(* Logix 5000 project; controller Commerford_topping_5477_V3 vendor 1 type 14 code 222 rev 33.11; software revision 33.02; part 2 of 6 *)
(* tags used below, declared in another part *)
   PackTags : PACKMLv30;
   Sts_Clearing : BOOL;   // Clearing
   Sts_Starting : BOOL;   // Starting
   Sts_Execute : BOOL;   // Execute
   Sts_Stopping : BOOL;   // Stopping
   Sts_Aborting : BOOL;   // Aborting
   Sts_Holding : BOOL;   // Holding
   Sts_Unholding : BOOL;   // Unholding
   Sts_Suspending : BOOL;   // Suspending
   Sts_Unsuspending : BOOL;   // Unsuspending
   Sts_Resetting : BOOL;   // Resetting
   Sts_Completing : BOOL;   // Completing
   Process_Selected : SINT;   // Recipe number selects which PackTag.command.product[#] will be used.
   Sts_MachineFaulted : BOOL;   // Machine recieved an fault trigger
   Sts_ProcessActive : BOOL;   // Machine is running a process.
   Reset_Signal : BOOL;   // Reset signal to EMs
   MachineState : USINT;   // Technical Report Equipment States: 1 Clearing 2 Stopped 3 Starting 4 Idle 5 Suspended 6 Execute 7 Stopping 8 Aborting 9
   wrk_compare_UDINT : UDINT;
   i : DINT;   // index num, only for local use. used for forloops
   wrk_prev_state : DINT;   // local mem
   wrk_SwitchLayer_To_Maintenance : DINT;
   wrk_SwitchLayer_To_Manual : DINT;
   wrk_SwitchLayer_To_Automatic : DINT;
(* ISA_TR_88_00_02, continued *)

ROUTINE Prescan   (* structured text *)
// Clear old mem
   ////////////////////////////////////////////////////////////
   //   Copyright (c)
   //------------------------------------------------------------
   //   Routine: Prescan
   //   Author: WPI\tom.reit
   //   Created: 2-11-2022
   //------------------------------------------------------------
   //   Description:
   //           Clear old mem
   //
   //
   //   History:
   //
   ////////////////////////////////////////////////////////////
   
   wrk_compare_UDINT:=0;
   for i := 0 to 31 do
   	wrk_compare_UDINT:=(1*2**i)+wrk_compare_UDINT;	// set compare value, cant move 64bits so have to do some clever bit manipulation.
   end_for;
   
   
   wrk_prev_state						:=	-1;					// set mem state to something that machineState can never be. therfor the whileloop will always execute
   MachineState						:=	9;					// always start safe, in aborted.
   Sts_MachineFaulted					:=	1;					// Machine is always faulted on startup from cold start.
   PackTags.Status.StateRequested		:=	MachineState;		// Set requested state same as actual state.
   
   wrk_SwitchLayer_To_Maintenance		:=0;		// Set layer switching to begin step.
   wrk_SwitchLayer_To_Manual			:=0;		// Set layer switching to begin step.
   wrk_SwitchLayer_To_Automatic		:=0;		// Set layer switching to begin step.
   
   Process_Selected					:=1;		// always run with first recipe on start.
   
   /* Reset ModeCumulativeTime for admin tags */
   for i := 0 to 6 do
   	PackTags.Admin.ModeCumulativeTime[i]:=0;
   end_for;
   
   Sts_ProcessActive:=0;
   
END_ROUTINE
END_ADD_ON_INSTRUCTION

ADD_ON_INSTRUCTION ISA_TR_88_00_02_StateChangeRequest   (* revision 1.0, ExecutePrescan, ExecuteEnableInFalse *)
VAR_IN_OUT
   Packml : PACKMLv30; {required}
END_VAR
VAR_INPUT
   RequestCmd : USINT; {required}   // 0 Undefined 1 Reset 2 Start 3 Stop 4 Hold 5 Unhold 6 Suspend 7 Unsuspend 8 Abort 9 Clear
END_VAR
VAR_OUTPUT
   Sts_StateTransition_Succesfull : BOOL; {access Read Only, visible}
   Sts_StateTransition_Failed : BOOL; {access Read Only, visible}
END_VAR
VAR
   dstepnum : DINT; {access None}
   Wrk_requestedState : DINT; {access None}
   ValidRequest : BOOL; {access None}   // check if request is valid
END_VAR

ROUTINE EnableInFalse   (* structured text *)
   ////////////////////////////////////////////////////////////
   //   Copyright (c)
   //------------------------------------------------------------
   //   Routine: EnableInFalse
   //   Author: WPI\tom.reit
   //   Created: 25-5-2023
   //------------------------------------------------------------
   //   Description:
   //
   //
   //   History:
   //
   ////////////////////////////////////////////////////////////
   dstepnum							:=0;
   Sts_StateTransition_Succesfull		:=0;
   Sts_StateTransition_Failed			:=0;
END_ROUTINE

ROUTINE Logic   (* structured text *)
   ////////////////////////////////////////////////////////////
   //   Copyright (c)
   //------------------------------------------------------------
   //   Routine: ISA_TR_88_00_02_StateChangeRequest - Logic
   //   Author: WPI\tom.reit
   //   Created: 24-5-2023
   //------------------------------------------------------------
   //   Description:
   //
   //
   //   History:
   //
   ////////////////////////////////////////////////////////////
   if dstepnum=0 AND EnableIn then
   	Sts_StateTransition_Succesfull		:=0;
   	Sts_StateTransition_Failed			:=0;
   	dstepnum:=1;
   end_if;
   case dstepnum of
   	1: /* send Unit command */
   		ValidRequest					:=0;
   		Packml.Command.CntrlCmd			:=RequestCmd;
   		Packml.Command.CmdChangeRequest	:=1;
   		case RequestCmd of
   			0:/* Undefined */
   			1:/* Reset */
   				if Packml.Status.StateCurrent = 2 then ValidRequest:=1; end_if;
   			2:/* Start */
   				if Packml.Status.StateCurrent = 4 then ValidRequest:=1; end_if;
   			3:/* Stop */
   				if Packml.Status.StateCurrent <> 8 then ValidRequest:=1; end_if;
   				if Packml.Status.StateCurrent <> 9 then ValidRequest:=1; end_if;
   				if Packml.Status.StateCurrent <> 1 then ValidRequest:=1; end_if;
   			4:/* Hold */
   				if Packml.Status.StateCurrent = 6 then ValidRequest:=1; end_if;
   			5:/* Unhold */
   				if Packml.Status.StateCurrent = 11 then ValidRequest:=1; end_if;
   			6:/* Suspend */
   				if Packml.Status.StateCurrent = 6 then ValidRequest:=1; end_if;
   			7:/* Unsuspend */
   				if Packml.Status.StateCurrent = 5 then ValidRequest:=1; end_if;
   			8:/* Abort */
   				ValidRequest:=1;
   			9:/* Clear */
   				if Packml.Status.StateCurrent = 9 then ValidRequest:=1; end_if;
   			10:/* Complete */
   				if Packml.Status.StateCurrent = 6 then ValidRequest:=1; end_if;
   			else
   		end_case;
   		dstepnum						:=2;
   	2: /* Acknowledge Unit Status, machine recieved command. */
   		if ValidRequest then
   			dstepnum						:=3;
   		else
   			dstepnum						:=999;
   		end_if;
   	3: /* Acknowledge Unit Status, machine recieved command. */
   		if NOT Packml.Command.CmdChangeRequest then
   			dstepnum						:=1000;
   		end_if;
   	999:/* Failed */
   		Sts_StateTransition_Succesfull		:=0;
   		Sts_StateTransition_Failed			:=1;
   	1000:/* Succesfull */
   		Sts_StateTransition_Succesfull		:=1;
   		Sts_StateTransition_Failed			:=0;
   	else
   		dstepnum:=0;
   end_case;
   
END_ROUTINE

ROUTINE Prescan   (* structured text *)
   ////////////////////////////////////////////////////////////
   //   Copyright (c)
   //------------------------------------------------------------
   //   Routine: Prescan
   //   Author: WPI\tom.reit
   //   Created: 25-5-2023
   //------------------------------------------------------------
   //   Description:
   //
   //
   //   History:
   //
   ////////////////////////////////////////////////////////////
   dstepnum							:=0;
   Sts_StateTransition_Succesfull		:=0;
   Sts_StateTransition_Failed			:=0;
END_ROUTINE
END_ADD_ON_INSTRUCTION

ADD_ON_INSTRUCTION ProcessHandler   (* revision 1.0, vendor WPI *)
VAR_IN_OUT
   PackML : ISA_TR_88_00_02; {required}
   bStateTransitions : DINT[32]; {required}
END_VAR
VAR_OUTPUT
   Sts_Unsuspending_PC : BOOL; {access Read Only}
   Sts_Unholding_PC : BOOL; {access Read Only}
   Sts_SuspendTrigger : BOOL; {access Read Only}
   Sts_Suspending_PC : BOOL; {access Read Only}
   Sts_Stopping_PC : BOOL; {access Read Only}
   Sts_Starting_PC : BOOL; {access Read Only}
   Sts_Resetting_PC : BOOL; {access Read Only}
   Sts_Holding_PC : BOOL; {access Read Only}
   Sts_Force_Stop : BOOL; {access Read Only}
   Sts_Force_Abort : BOOL; {access Read Only}
   Sts_Faulted : BOOL; {access Read Only}
   Sts_Executing : BOOL; {access Read Only}
   Sts_Process_Selected : BOOL; {access Read Only, visible}
   Sts_Completing_PC : BOOL; {access Read Only}
   Sts_Clearing_PC : BOOL; {access Read Only}
   Sts_Aborting_PC : BOOL; {access Read Only}
   OwnershipFault : BOOL; {access Read Only, visible}
END_VAR
VAR_INPUT
   Select : BOOL; {visible}   // Selecting Process will incuding in Unit state transitions
END_VAR
VAR_IN_OUT
   ProcessModule : ProcessModule; {required}
END_VAR
VAR_INPUT
   Process_ID : USINT; {required}
END_VAR
VAR
   UnasignOwnership : BOOL; {access None}
   AsignOwnership : BOOL; {access None}
END_VAR

ROUTINE Logic   (* ladder *)
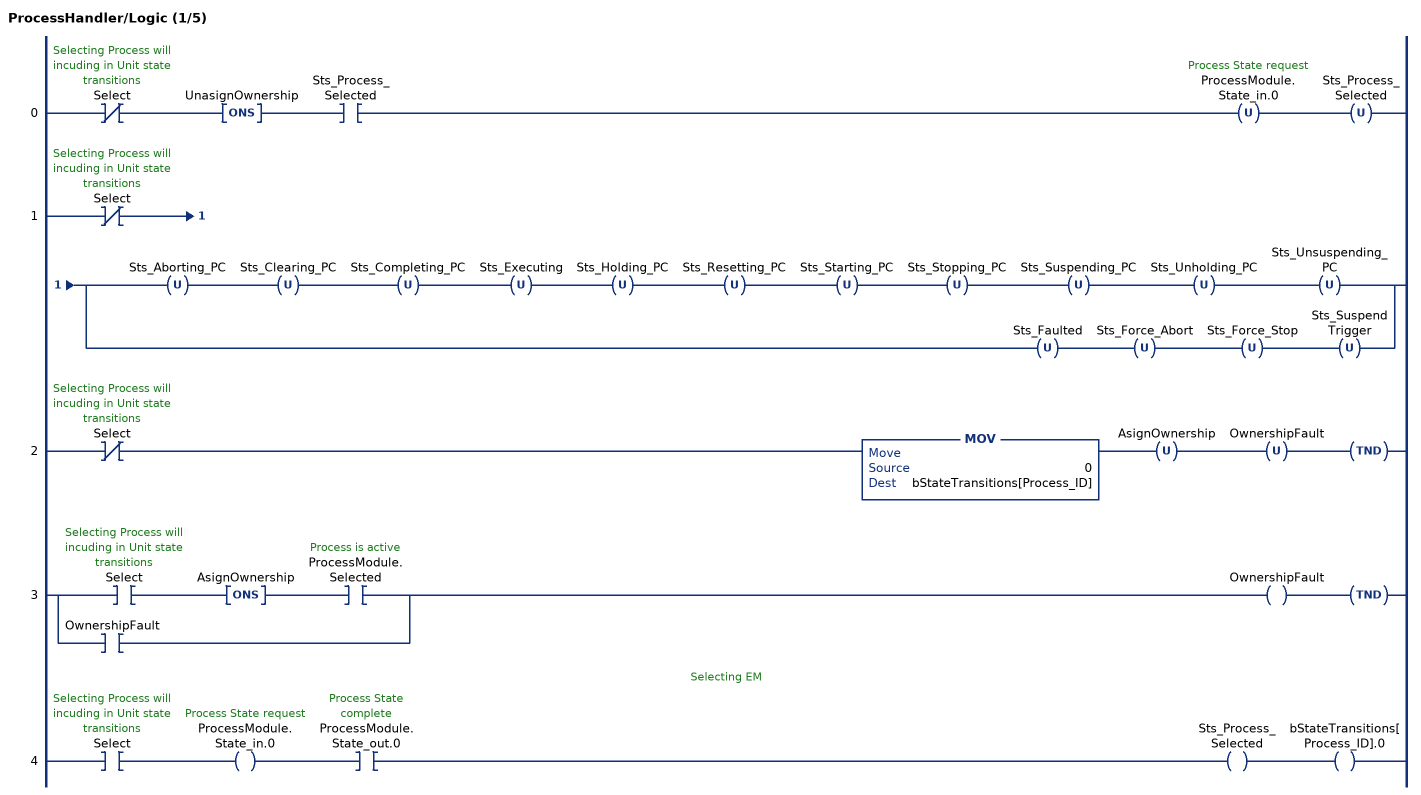
   0: XIO(Select)ONS(UnasignOwnership)XIC(Sts_Process_Selected)OTU(ProcessModule.State_in.0)OTU(Sts_Process_Selected);
   1: XIO(Select)[OTU(Sts_Aborting_PC) OTU(Sts_Clearing_PC) OTU(Sts_Completing_PC) OTU(Sts_Executing) OTU(Sts_Holding_PC) OTU(Sts_Resetting_PC) OTU(Sts_Starting_PC) OTU(Sts_Stopping_PC) OTU(Sts_Suspending_PC) OTU(Sts_Unholding_PC) OTU(Sts_Unsuspending_PC) ,OTU(Sts_Faulted) OTU(Sts_Force_Abort) OTU(Sts_Force_Stop) OTU(Sts_SuspendTrigger) ];
   2: XIO(Select)MOV(0,bStateTransitions[Process_ID])OTU(AsignOwnership)OTU(OwnershipFault)TND();
   3: [XIC(Select) ONS(AsignOwnership) XIC(ProcessModule.Selected) ,XIC(OwnershipFault) ]OTE(OwnershipFault)TND();
   // Selecting EM
   4: XIC(Select)OTE(ProcessModule.State_in.0)XIC(ProcessModule.State_out.0)OTE(Sts_Process_Selected)OTE(bStateTransitions[Process_ID].0);
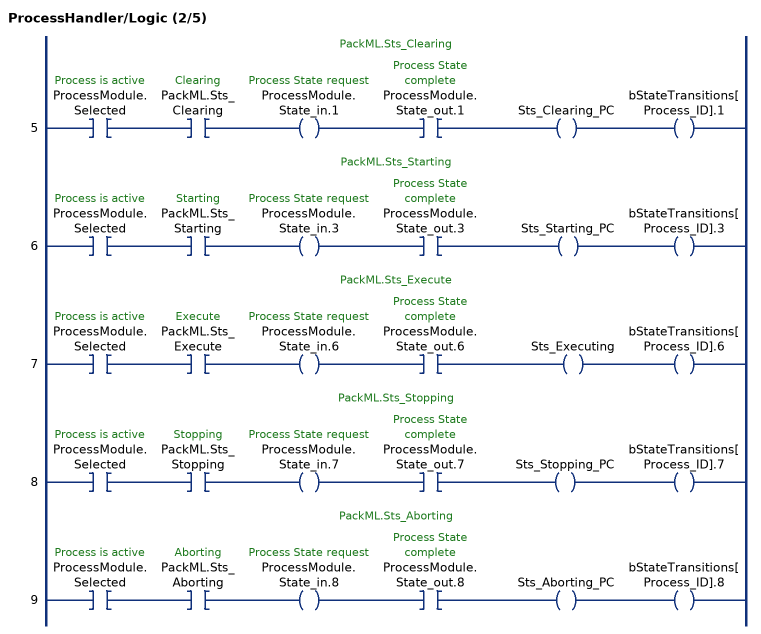
   // PackML.Sts_Clearing
   5: XIC(ProcessModule.Selected)XIC(PackML.Sts_Clearing)OTE(ProcessModule.State_in.1)XIC(ProcessModule.State_out.1)OTE(Sts_Clearing_PC)OTE(bStateTransitions[Process_ID].1);
   // PackML.Sts_Starting
   6: XIC(ProcessModule.Selected)XIC(PackML.Sts_Starting)OTE(ProcessModule.State_in.3)XIC(ProcessModule.State_out.3)OTE(Sts_Starting_PC)OTE(bStateTransitions[Process_ID].3);
   // PackML.Sts_Execute
   7: XIC(ProcessModule.Selected)XIC(PackML.Sts_Execute)OTE(ProcessModule.State_in.6)XIC(ProcessModule.State_out.6)OTE(Sts_Executing)OTE(bStateTransitions[Process_ID].6);
   // PackML.Sts_Stopping
   8: XIC(ProcessModule.Selected)XIC(PackML.Sts_Stopping)OTE(ProcessModule.State_in.7)XIC(ProcessModule.State_out.7)OTE(Sts_Stopping_PC)OTE(bStateTransitions[Process_ID].7);
   // PackML.Sts_Aborting
   9: XIC(ProcessModule.Selected)XIC(PackML.Sts_Aborting)OTE(ProcessModule.State_in.8)XIC(ProcessModule.State_out.8)OTE(Sts_Aborting_PC)OTE(bStateTransitions[Process_ID].8);
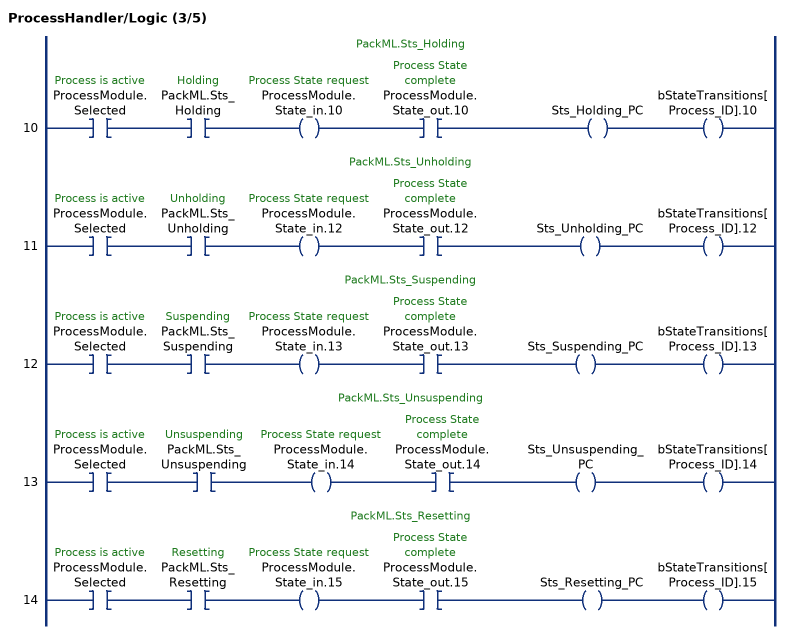
   // PackML.Sts_Holding
   10: XIC(ProcessModule.Selected)XIC(PackML.Sts_Holding)OTE(ProcessModule.State_in.10)XIC(ProcessModule.State_out.10)OTE(Sts_Holding_PC)OTE(bStateTransitions[Process_ID].10);
   // PackML.Sts_Unholding
   11: XIC(ProcessModule.Selected)XIC(PackML.Sts_Unholding)OTE(ProcessModule.State_in.12)XIC(ProcessModule.State_out.12)OTE(Sts_Unholding_PC)OTE(bStateTransitions[Process_ID].12);
   // PackML.Sts_Suspending
   12: XIC(ProcessModule.Selected)XIC(PackML.Sts_Suspending)OTE(ProcessModule.State_in.13)XIC(ProcessModule.State_out.13)OTE(Sts_Suspending_PC)OTE(bStateTransitions[Process_ID].13);
   // PackML.Sts_Unsuspending
   13: XIC(ProcessModule.Selected)XIC(PackML.Sts_Unsuspending)OTE(ProcessModule.State_in.14)XIC(ProcessModule.State_out.14)OTE(Sts_Unsuspending_PC)OTE(bStateTransitions[Process_ID].14);
   // PackML.Sts_Resetting
   14: XIC(ProcessModule.Selected)XIC(PackML.Sts_Resetting)OTE(ProcessModule.State_in.15)XIC(ProcessModule.State_out.15)OTE(Sts_Resetting_PC)OTE(bStateTransitions[Process_ID].15);
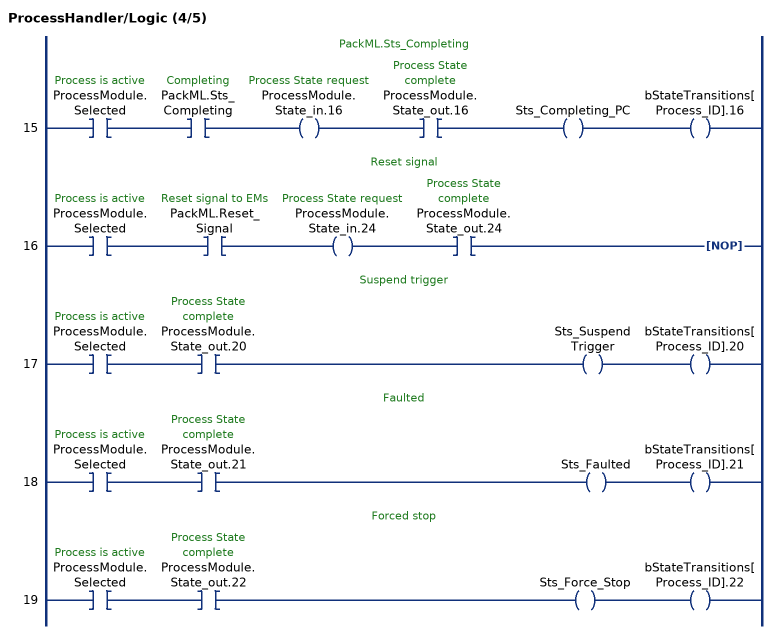
   // PackML.Sts_Completing
   15: XIC(ProcessModule.Selected)XIC(PackML.Sts_Completing)OTE(ProcessModule.State_in.16)XIC(ProcessModule.State_out.16)OTE(Sts_Completing_PC)OTE(bStateTransitions[Process_ID].16);
   // Reset signal
   16: XIC(ProcessModule.Selected)XIC(PackML.Reset_Signal)OTE(ProcessModule.State_in.24)XIC(ProcessModule.State_out.24)NOP();
   // Suspend trigger
   17: XIC(ProcessModule.Selected)XIC(ProcessModule.State_out.20)OTE(Sts_SuspendTrigger)OTE(bStateTransitions[Process_ID].20);
   // Faulted
   18: XIC(ProcessModule.Selected)XIC(ProcessModule.State_out.21)OTE(Sts_Faulted)OTE(bStateTransitions[Process_ID].21);
   // Forced stop
   19: XIC(ProcessModule.Selected)XIC(ProcessModule.State_out.22)OTE(Sts_Force_Stop)OTE(bStateTransitions[Process_ID].22);
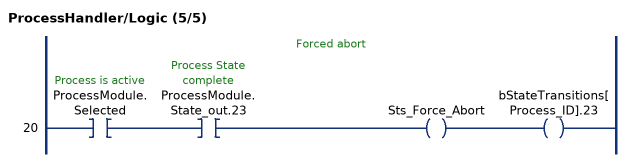
   // Forced abort
   20: XIC(ProcessModule.Selected)XIC(ProcessModule.State_out.23)OTE(Sts_Force_Abort)OTE(bStateTransitions[Process_ID].23);
END_ROUTINE
END_ADD_ON_INSTRUCTION

VAR_GLOBAL   (* controller tags *)
   HMI_SAF_Reset : BOOL;   // Safety reset for HMI
END_VAR

PROGRAM MainProgram   (* main routine MainRoutine *)

ROUTINE MainRoutine   (* ladder *)
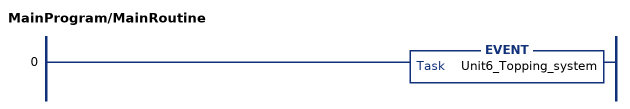
   0: EVENT(Unit6_Topping_system);
END_ROUTINE
END_PROGRAM

PROGRAM SafetyProgram   (* main routine MainRoutine, safety *)

ROUTINE MainRoutine   (* ladder *)
END_ROUTINE
END_PROGRAM

PROGRAM UN6_EM1_Buffertank   (* main routine Main *)
// Buffertank, generated by G.E.M
VAR
   _Cmd_Activate : BOOL;
   _Cmd_ClearFaults : BOOL;
   _Cmd_Deactivate : BOOL;
   _Cmd_Reset : BOOL;
   _Sts_AcivateSeq_PC : BOOL;
   _Sts_ClearSeq_PC : BOOL;
   _Sts_DeactivateSeq_PC : BOOL;
   _Sts_Execute_PC : BOOL;
   _Sts_ResetSeq_PC : BOOL;
END_VAR
VAR {public}
   EquipmentModule : EquipmentModule := (Selected := 1, State_in := 2#0000_0000_0000_0000_0000_0000_0000_0101, State_out := 2#0000_0000_0000_0000_0000_0000_0000_0001, _SEQ.Clearing := -1, _SEQ.Activating := -1, _SEQ.Deactivating := -1, _SEQ.Resetting := -1);
        .State_in.1   // Clearing
END_VAR

ROUTINE _EP_Acivate   (* ladder *)
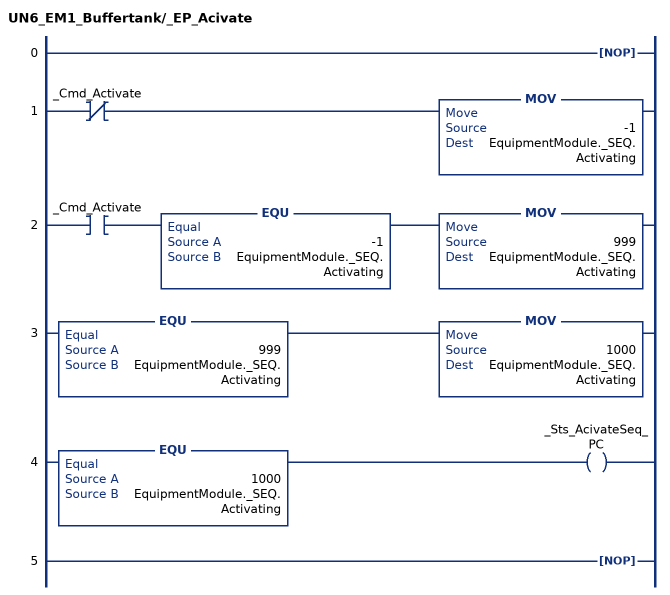
   0: NOP();
   1: XIO(_Cmd_Activate)MOV(-1,EquipmentModule._SEQ.Activating);
   2: XIC(_Cmd_Activate)EQU(-1,EquipmentModule._SEQ.Activating)MOV(999,EquipmentModule._SEQ.Activating);
   3: EQU(999,EquipmentModule._SEQ.Activating)MOV(1000,EquipmentModule._SEQ.Activating);
   4: EQU(1000,EquipmentModule._SEQ.Activating)OTE(_Sts_AcivateSeq_PC);
   5: NOP();
END_ROUTINE

ROUTINE _EP_Clear   (* ladder *)
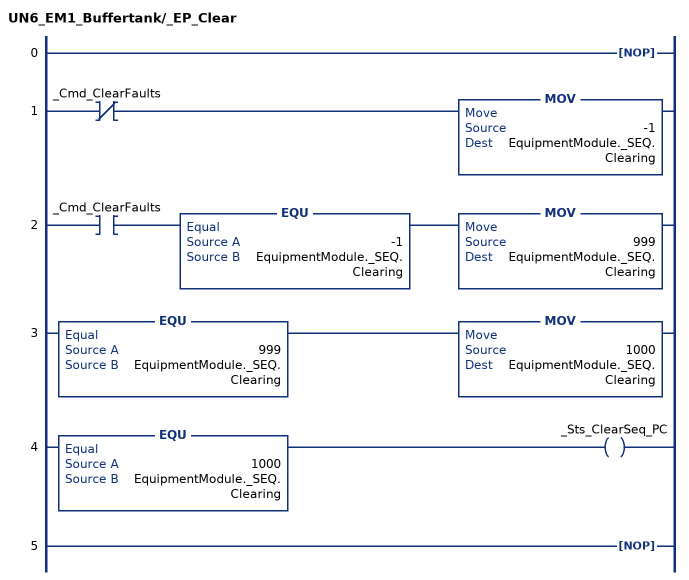
   0: NOP();
   1: XIO(_Cmd_ClearFaults)MOV(-1,EquipmentModule._SEQ.Clearing);
   2: XIC(_Cmd_ClearFaults)EQU(-1,EquipmentModule._SEQ.Clearing)MOV(999,EquipmentModule._SEQ.Clearing);
   3: EQU(999,EquipmentModule._SEQ.Clearing)MOV(1000,EquipmentModule._SEQ.Clearing);
   4: EQU(1000,EquipmentModule._SEQ.Clearing)OTE(_Sts_ClearSeq_PC);
   5: NOP();
END_ROUTINE

ROUTINE _EP_Deactivate   (* ladder *)
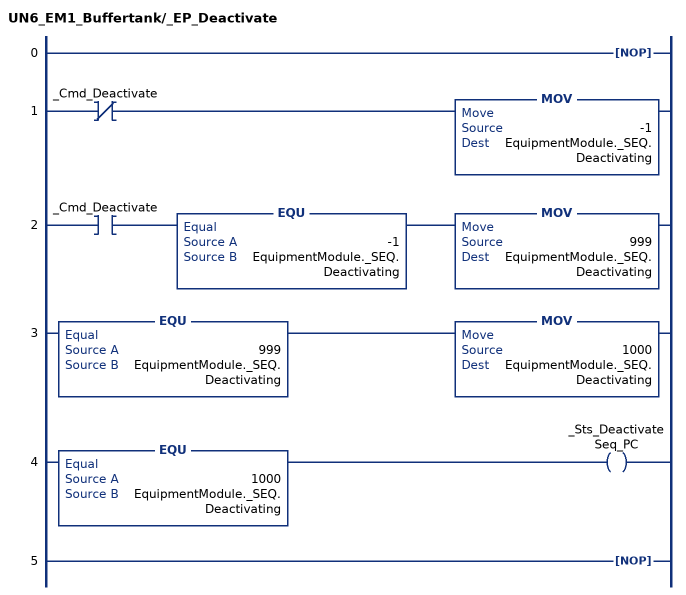
   0: NOP();
   1: XIO(_Cmd_Deactivate)MOV(-1,EquipmentModule._SEQ.Deactivating);
   2: XIC(_Cmd_Deactivate)EQU(-1,EquipmentModule._SEQ.Deactivating)MOV(999,EquipmentModule._SEQ.Deactivating);
   3: EQU(999,EquipmentModule._SEQ.Deactivating)MOV(1000,EquipmentModule._SEQ.Deactivating);
   4: EQU(1000,EquipmentModule._SEQ.Deactivating)OTE(_Sts_DeactivateSeq_PC);
   5: NOP();
END_ROUTINE

ROUTINE _EP_Resetting   (* ladder *)
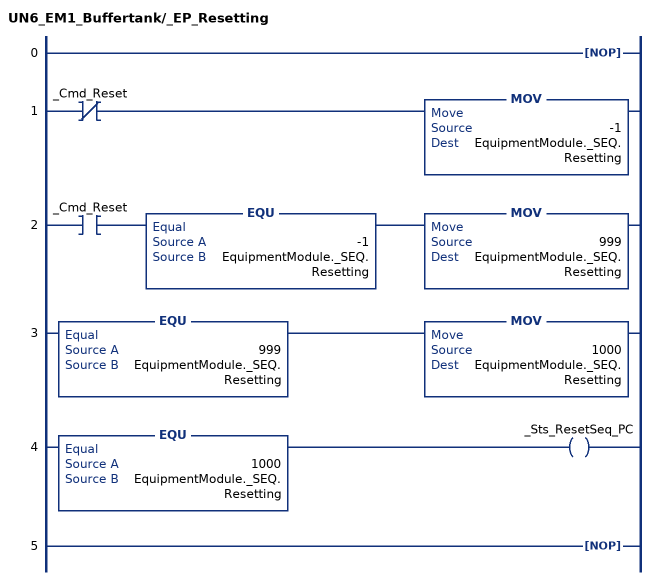
   0: NOP();
   1: XIO(_Cmd_Reset)MOV(-1,EquipmentModule._SEQ.Resetting);
   2: XIC(_Cmd_Reset)EQU(-1,EquipmentModule._SEQ.Resetting)MOV(999,EquipmentModule._SEQ.Resetting);
   3: EQU(999,EquipmentModule._SEQ.Resetting)MOV(1000,EquipmentModule._SEQ.Resetting);
   4: EQU(1000,EquipmentModule._SEQ.Resetting)OTE(_Sts_ResetSeq_PC);
   5: NOP();
END_ROUTINE

ROUTINE _EP_Running   (* ladder *)
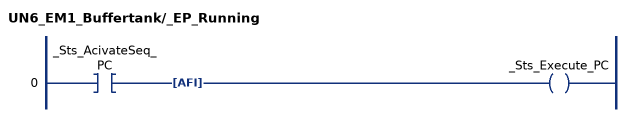
   0: XIC(_Sts_AcivateSeq_PC)AFI()OTE(_Sts_Execute_PC);
END_ROUTINE

ROUTINE _FaultHandler   (* ladder *)
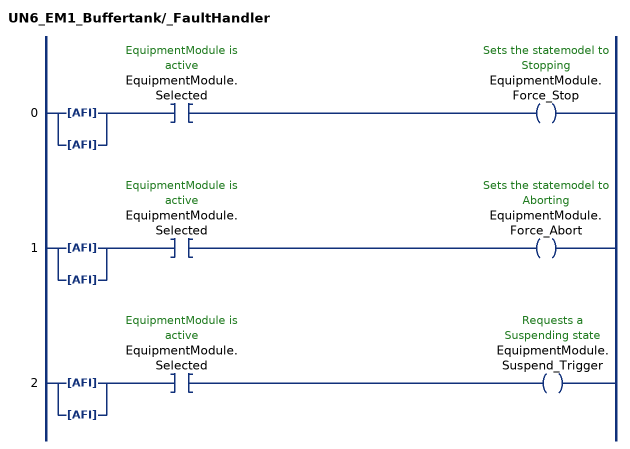
   0: [AFI() ,AFI() ]XIC(EquipmentModule.Selected)OTE(EquipmentModule.Force_Stop);
   1: [AFI() ,AFI() ]XIC(EquipmentModule.Selected)OTE(EquipmentModule.Force_Abort);
   2: [AFI() ,AFI() ]XIC(EquipmentModule.Selected)OTE(EquipmentModule.Suspend_Trigger);
END_ROUTINE

ROUTINE _INOUT   (* ladder *)
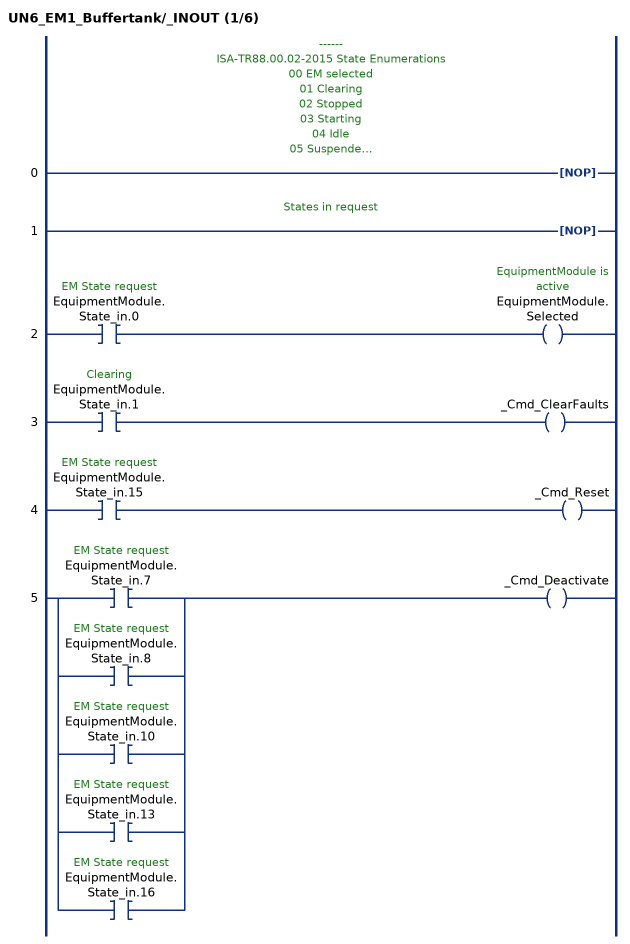
   // ------
   // ISA-TR88.00.02-2015 State Enumerations
   // 00 EM selected
   // 01 Clearing
   // 02 Stopped
   // 03 Starting
   // 04 Idle
   // 05 Suspended
   // 06 Execute
   // 07 Stopping
   // 08 Aborting
   // 09 Aborted
   // 10 Holding
   // 11 Held
   // 12 UnHolding
   // 13 Suspending
   // 14 Unsuspending
   // 15 Resetting
   // 16 Completing
   // 17 Complete
   // 18 Undefined
   // 19 Undefined
   // 20 Suspend trigger
   // 21 Faulted
   // 22 Force stop
   // 23 Force abort
   // 24 Reset signal
   // 31 Undefined
   // ------
   0: NOP();
   // States in request
   1: NOP();
   2: XIC(EquipmentModule.State_in.0)OTE(EquipmentModule.Selected);
   3: XIC(EquipmentModule.State_in.1)OTE(_Cmd_ClearFaults);
   4: XIC(EquipmentModule.State_in.15)OTE(_Cmd_Reset);
   5: [XIC(EquipmentModule.State_in.7) ,XIC(EquipmentModule.State_in.8) ,XIC(EquipmentModule.State_in.10) ,XIC(EquipmentModule.State_in.13) ,XIC(EquipmentModule.State_in.16) ]OTE(_Cmd_Deactivate);
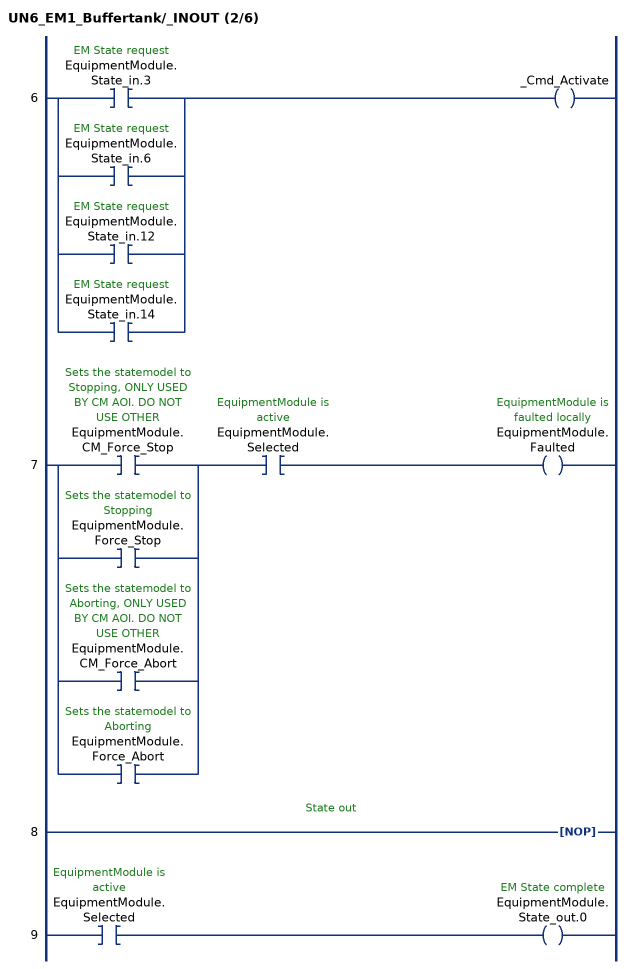
   6: [XIC(EquipmentModule.State_in.3) ,XIC(EquipmentModule.State_in.6) ,XIC(EquipmentModule.State_in.12) ,XIC(EquipmentModule.State_in.14) ]OTE(_Cmd_Activate);
   7: [XIC(EquipmentModule.CM_Force_Stop) ,XIC(EquipmentModule.Force_Stop) ,XIC(EquipmentModule.CM_Force_Abort) ,XIC(EquipmentModule.Force_Abort) ]XIC(EquipmentModule.Selected)OTE(EquipmentModule.Faulted);
   // State out
   8: NOP();
   9: XIC(EquipmentModule.Selected)OTE(EquipmentModule.State_out.0);
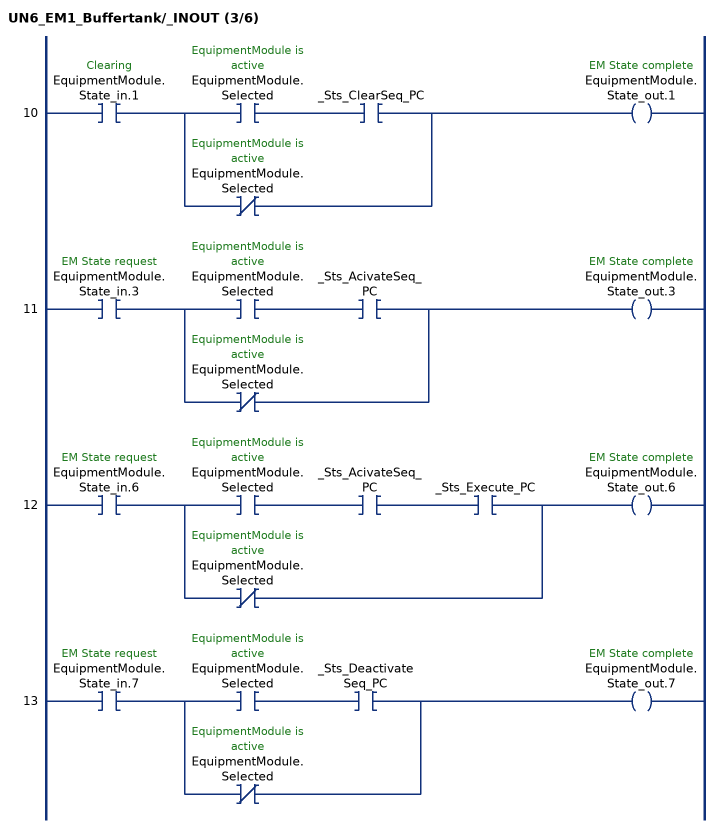
   10: XIC(EquipmentModule.State_in.1)[XIC(EquipmentModule.Selected) XIC(_Sts_ClearSeq_PC) ,XIO(EquipmentModule.Selected) ]OTE(EquipmentModule.State_out.1);
   11: XIC(EquipmentModule.State_in.3)[XIC(EquipmentModule.Selected) XIC(_Sts_AcivateSeq_PC) ,XIO(EquipmentModule.Selected) ]OTE(EquipmentModule.State_out.3);
   12: XIC(EquipmentModule.State_in.6)[XIC(EquipmentModule.Selected) XIC(_Sts_AcivateSeq_PC) XIC(_Sts_Execute_PC) ,XIO(EquipmentModule.Selected) ]OTE(EquipmentModule.State_out.6);
   13: XIC(EquipmentModule.State_in.7)[XIC(EquipmentModule.Selected) XIC(_Sts_DeactivateSeq_PC) ,XIO(EquipmentModule.Selected) ]OTE(EquipmentModule.State_out.7);
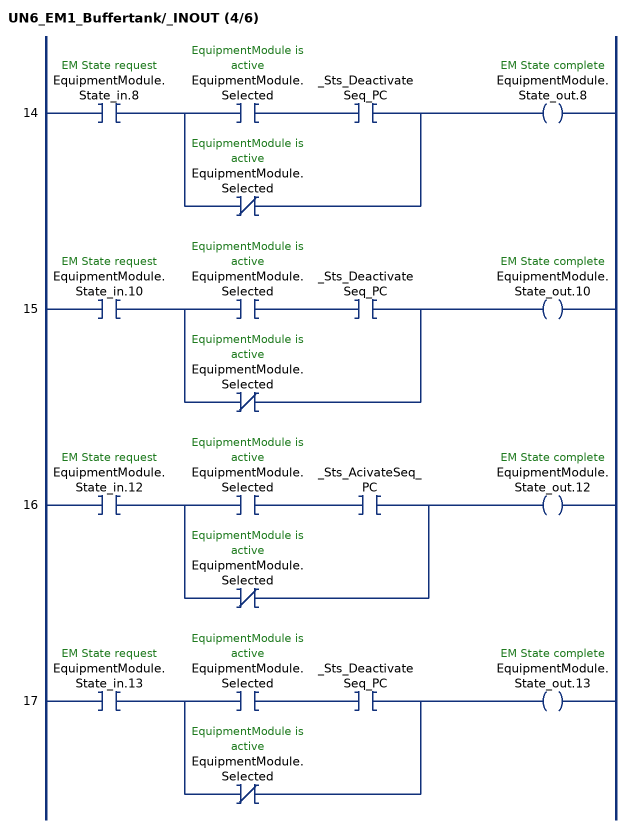
   14: XIC(EquipmentModule.State_in.8)[XIC(EquipmentModule.Selected) XIC(_Sts_DeactivateSeq_PC) ,XIO(EquipmentModule.Selected) ]OTE(EquipmentModule.State_out.8);
   15: XIC(EquipmentModule.State_in.10)[XIC(EquipmentModule.Selected) XIC(_Sts_DeactivateSeq_PC) ,XIO(EquipmentModule.Selected) ]OTE(EquipmentModule.State_out.10);
   16: XIC(EquipmentModule.State_in.12)[XIC(EquipmentModule.Selected) XIC(_Sts_AcivateSeq_PC) ,XIO(EquipmentModule.Selected) ]OTE(EquipmentModule.State_out.12);
   17: XIC(EquipmentModule.State_in.13)[XIC(EquipmentModule.Selected) XIC(_Sts_DeactivateSeq_PC) ,XIO(EquipmentModule.Selected) ]OTE(EquipmentModule.State_out.13);
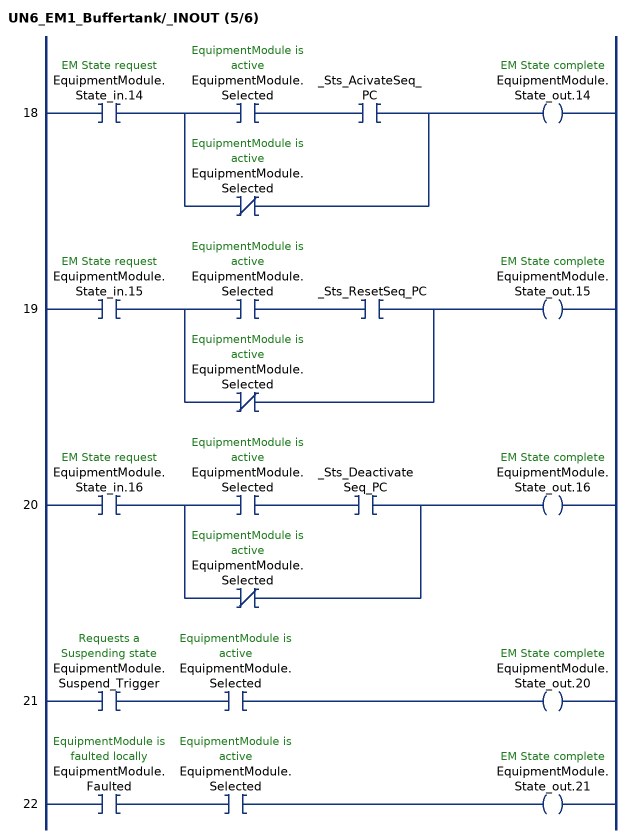
   18: XIC(EquipmentModule.State_in.14)[XIC(EquipmentModule.Selected) XIC(_Sts_AcivateSeq_PC) ,XIO(EquipmentModule.Selected) ]OTE(EquipmentModule.State_out.14);
   19: XIC(EquipmentModule.State_in.15)[XIC(EquipmentModule.Selected) XIC(_Sts_ResetSeq_PC) ,XIO(EquipmentModule.Selected) ]OTE(EquipmentModule.State_out.15);
   20: XIC(EquipmentModule.State_in.16)[XIC(EquipmentModule.Selected) XIC(_Sts_DeactivateSeq_PC) ,XIO(EquipmentModule.Selected) ]OTE(EquipmentModule.State_out.16);
   21: XIC(EquipmentModule.Suspend_Trigger)XIC(EquipmentModule.Selected)OTE(EquipmentModule.State_out.20);
   22: XIC(EquipmentModule.Faulted)XIC(EquipmentModule.Selected)OTE(EquipmentModule.State_out.21);
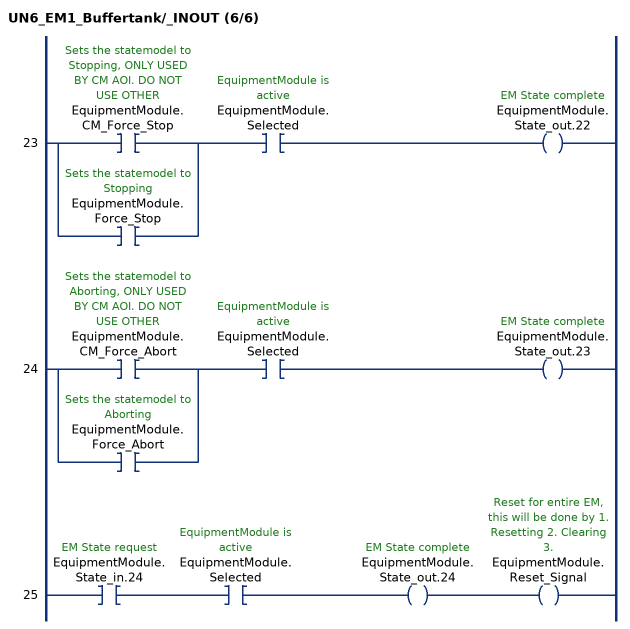
   23: [XIC(EquipmentModule.CM_Force_Stop) ,XIC(EquipmentModule.Force_Stop) ]XIC(EquipmentModule.Selected)OTE(EquipmentModule.State_out.22);
   24: [XIC(EquipmentModule.CM_Force_Abort) ,XIC(EquipmentModule.Force_Abort) ]XIC(EquipmentModule.Selected)OTE(EquipmentModule.State_out.23);
   25: XIC(EquipmentModule.State_in.24)XIC(EquipmentModule.Selected)OTE(EquipmentModule.State_out.24)OTE(EquipmentModule.Reset_Signal);
END_ROUTINE
